INTERFACE I_AsyncRpcCall EXTENDS I_Disposable

METHOD PUBLIC Call
VAR_INPUT
END_VAR
END_METHOD

END_INTERFACE

(* stored: Version 1.1.0.1, ProductVersion 3.1.4024.12
   Itf I_AsyncRpcCall: Id {9081126a-e6e8-4e68-b982-e20ff71f1cb5}
   Method Call: Id {ece72c8e-fd90-46a1-8855-728fd24ec460} *)
